FUNCTION_BLOCK PT1 (* discrete PT1 low-pass filter *)
  (* Standard: 61499-2 *)
  (* Version 1.0, 2026-04-22, Thomas Mayr *)
  PACKAGE eclipse4diac::signalprocessing;
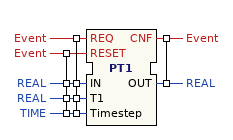
  EVENT_INPUT
    REQ WITH IN, T1, Timestep; (* Calculate next output *)
    RESET WITH IN, T1, Timestep; (* Reset internal filter state *)
  END_EVENT
  EVENT_OUTPUT
    CNF WITH OUT; (* Output value updated *)
  END_EVENT
  VAR_INPUT
    IN : REAL; (* Input value *)
    T1 : REAL; (* PT1 time constant [s] *)
    Timestep : TIME; (* Sampling time *)
  END_VAR
  VAR_OUTPUT
    OUT : REAL; (* Filtered output value *)
  END_VAR
  VAR
    alpha : REAL;
    state : REAL;
    initialized : BOOL;
    DT_SEC : REAL;
  END_VAR
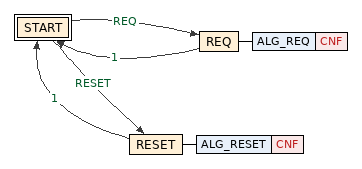
  EC_STATES
    START; (* Initial State *)
    REQ : ALG_REQ -> CNF;
    RESET : ALG_RESET -> CNF;
  END_STATES
  EC_TRANSITIONS
    START TO REQ := REQ;
    REQ TO START := 1;
    START TO RESET := RESET;
    RESET TO START := 1;
  END_TRANSITIONS
  ALGORITHM ALG_REQ IN ST:
DT_SEC := LREAL_TO_REAL(TIME_IN_S_TO_LREAL(Timestep));
IF DT_SEC <= 0.0 THEN
	OUT := IN;
	state := OUT;
	initialized := TRUE;
	RETURN;
END_IF;

IF T1 <= 0.0 THEN
	OUT := IN;
	state := OUT;
	initialized := TRUE;
	RETURN;
END_IF;

alpha := DT_SEC / (T1 + DT_SEC);

IF NOT initialized THEN
	state := IN;
	initialized := TRUE;
ELSE
	state := state + alpha * (IN - state);
END_IF;

OUT := state;
  END_ALGORITHM
  ALGORITHM ALG_RESET IN ST:
state := 0.0;
alpha := 0.0;
initialized := FALSE;
OUT := 0.0;
  END_ALGORITHM
END_FUNCTION_BLOCK
